VAR_OUTPUT
	stErr : ST_SiftError;
END_VAR

IF pJsonBuffer = 0 THEN
	stErr.bError := TRUE;
	stErr.nErrId := GVL_SIFT.NULL_JSON_POINTER;
	stErr.sReason := 'The JSON buffer is null';
	RETURN;
END_IF

fbJson.StartObject();

fbJson.AddKey('api_key');
fbJson.AddString(sApiKey);

fbJson.AddKey('grpc_uri');
fbJson.AddString(sGrpcUri);

fbJson.EndObject();

pJsonString := pJsonBuffer;
nBytes := fbJson.CopyDocument(pJsonString^, nLength);
IF nBytes = 0 THEN
	stErr.nErrId := GVL_SIFT.JSON_CAPACITY_REACHED;
	stErr.bError := TRUE;
	stErr.sReason := CONCAT(
		CONCAT('JSON msg too large: ', UDINT_TO_STRING(fbJson.GetDocumentLength())),
		' endpoint=authenticate',
	);
	RETURN;
END_IF

stErr := _F_CreateEndpointMessage(sEndpoint:='authenticate', 
								  pData:=pJsonString, 
								  nLength:=nBytes-1, 
                                  nBufferLength := nLength, 
                                  stMsg:=stMsg);

END_FUNCTION

// ---- POUs/Services/FB_PingService.TcPOU
FUNCTION_BLOCK FB_PingService
VAR_INPUT
	hSiftClient : T_SiftClient;
	bExecute : BOOL;
END_VAR

VAR_OUTPUT
	bBusy : BOOL;
	bError : BOOL;
	nErrId : UDINT;
	bSuccess : BOOL;
	stSiftError : ST_SiftError;
END_VAR

VAR
	eState : (IDLE, SEND_MESSAGE, WAIT_FOR_RESPONSE, SUCCESS, FAILURE) := IDLE;
	fbSendSiftMessage : _FB_SendSiftMessage;
	stPingReq : _ST_SiftMessage;
	fbJson : FB_JsonDomParser;
	sResponse : STRING(GVL_SIFT.MAX_JSON_RESPONSE_SIZE);
	jsonDoc : SJsonValue;
END_VAR

CASE eState OF
	IDLE:
		IF bExecute THEN
			eState := SEND_MESSAGE;
		END_IF
		
	SEND_MESSAGE:
		bBusy := TRUE;
		bError := FALSE;
		
		stSiftError := _F_CreatePingMessage(stMsg:=stPingReq);
		IF stSiftError.bError THEN
			nErrId := stSiftError.nErrId;
			eState := FAILURE;
		END_IF
		
		fbSendSiftMessage(hSiftClient:=hSiftClient, stMsg:=stPingReq, bExecute:=TRUE);
		eState := WAIT_FOR_RESPONSE;

	WAIT_FOR_RESPONSE:
		bBusy := TRUE;
		bError := FALSE;
		fbSendSiftMessage(bExecute:=FALSE);
		
		IF fbSendSiftMessage.bBusy THEN
			RETURN;
		ELSIF fbSendSiftMessage.bError THEN
			nErrId := GVL_SIFT.SIFT_PROXY_NO_RESPONSE;
			eState := FAILURE;
			RETURN;
		END_IF

		// Verify response.
		IF fbSendSiftMessage.stResponse.nLength > GVL_SIFT.MAX_JSON_RESPONSE_SIZE THEN
			nErrId := GVL_SIFT.JSON_CAPACITY_REACHED;
			eState := FAILURE;
			RETURN;	
		END_IF
		
		IF NOT SAFE_MEMCPY(ADR(sResponse), SIZEOF(sResponse), 
			               ADR(fbSendSiftMessage.stResponse.aData), fbSendSiftMessage.stResponse.nLength) THEN
			nErrId := GVL_SIFT.MEMCPY_ERROR;
			eState := FAILURE;
		END_IF
		
		jsonDoc := fbJson.ParseDocument(sResponse);
		
		IF _F_IsSuccessfulResponse(jsonDoc) THEN
			eState := SUCCESS;
		ELSE
			IF NOT _F_SetSiftError(jsonDoc, stSiftError) THEN
				nErrId := GVL_SIFT.SIFT_PROXY_INVALID_RESPONSE;
			END_IF
			nErrId := stSiftError.nErrId;
			eState := FAILURE;
		END_IF
		
	SUCCESS:
		bBusy := FALSE;
		bError := FALSE;
		bSuccess := TRUE;
		eState := IDLE;
		
	FAILURE:
		bBusy := FALSE;
		bError := TRUE;
		eState := IDLE;
END_CASE

END_FUNCTION_BLOCK

// ---- POUs/Services/FB_RunService.TcPOU
FUNCTION_BLOCK FB_RunService
VAR_INPUT
	hSiftClient : T_SiftClient;
	bExecute : BOOL;
	sName : STRING(255);
	sDescription : STRING(255);
	aTags : ARRAY[0..SiftClientParameters.MAX_NUM_TAGS - 1] OF STRING(255);
END_VAR

VAR_OUTPUT
	sId : STRING(255);
	bBusy : BOOL;
	bError : BOOL;
	nErrId : UDINT;
	stSiftError : ST_SiftError;
END_VAR

VAR
	eState : (IDLE, SEND_MESSAGE, WAIT_FOR_RESPONSE, SUCCESS, FAILURE) := IDLE;
	fbSendSiftMessage : _FB_SendSiftMessage;
	stRunReq : _ST_SiftMessage;
	fbJson : FB_JsonDomParser;
	sResponse : STRING(GVL_SIFT.MAX_JSON_RESPONSE_SIZE);
	jsonDoc : SJsonValue;	
END_VAR

CASE eState OF
	IDLE:
		IF bExecute THEN
			eState := SEND_MESSAGE;
		END_IF
		
	SEND_MESSAGE:
		bBusy := TRUE;
		bError := FALSE;
		
		stSiftError := _F_CreateRunMessage(stMsg:=stRunReq,
										   sName := sName,
										   sDescription := sDescription,
										   aTags := aTags,
										   pJsonBuffer := hSiftClient.pJsonBuffer,
										   nLength := hSiftClient.pJbLength);
		IF stSiftError.bError THEN
			nErrId := stSiftError.nErrId;
			eState := FAILURE;
		END_IF
		
		fbSendSiftMessage(hSiftClient:=hSiftClient, stMsg:=stRunReq, bExecute:=TRUE);
		eState := WAIT_FOR_RESPONSE;

	WAIT_FOR_RESPONSE:
		bBusy := TRUE;
		bError := FALSE;
		fbSendSiftMessage(bExecute := FALSE);
		
		IF fbSendSiftMessage.bBusy THEN
			RETURN;
		ELSIF fbSendSiftMessage.bError THEN
			nErrId := fbSendSiftMessage.nErrId;
			eState := FAILURE;
			RETURN;
		END_IF
		
		// Verify response.
		IF fbSendSiftMessage.stResponse.nLength > GVL_SIFT.MAX_JSON_RESPONSE_SIZE THEN
			nErrId := GVL_SIFT.JSON_CAPACITY_REACHED;
			eState := FAILURE;
			RETURN;	
		END_IF
		
		IF NOT SAFE_MEMCPY(ADR(sResponse), SIZEOF(sResponse), 
			               ADR(fbSendSiftMessage.stResponse.aData), fbSendSiftMessage.stResponse.nLength) THEN
			nErrId := GVL_SIFT.MEMCPY_ERROR;
			eState := FAILURE;
		END_IF
		
		jsonDoc := fbJson.ParseDocument(sResponse);
		IF jsonDoc = 0 THEN
			eState := FAILURE;
			nErrId := GVL_SIFT.UNABLE_TO_PARSE_JSON;
		END_IF
		
		IF _F_IsSuccessfulResponse(jsonDoc) THEN
			IF NOT fbJson.HasMember(jsonDoc, 'data') THEN
				nErrId := GVL_SIFT.SIFT_PROXY_INVALID_RESPONSE;
				eState := FAILURE;
				RETURN;
			END_IF
			jsonDoc := fbJson.FindMember(jsonDoc, 'data');
			
			IF NOT fbJson.HasMember(jsonDoc, 'run') THEN
				nErrId := GVL_SIFT.SIFT_PROXY_INVALID_RESPONSE;
				eState := FAILURE;
				RETURN;
			END_IF
			
			jsonDoc := fbJson.FindMember(jsonDoc, 'run');
			IF NOT fbJson.HasMember(jsonDoc, 'runId') THEN
				nErrId := GVL_SIFT.SIFT_PROXY_INVALID_RESPONSE;
				eState := FAILURE;
				RETURN;
			END_IF
			
			jsonDoc := fbJson.FindMember(jsonDoc, 'runId');
			sId := fbJson.GetString(jsonDoc);
			
			eState := SUCCESS;
		ELSE
			IF NOT _F_SetSiftError(jsonDoc, stSiftError) THEN
				nErrId := GVL_SIFT.SIFT_PROXY_INVALID_RESPONSE;
			END_IF
			nErrId := stSiftError.nErrId;
			eState := FAILURE;
		END_IF
		
	SUCCESS:
		bBusy := FALSE;
		bError := FALSE;
		eState := IDLE;
		
	FAILURE:
		bBusy := FALSE;
		bError := TRUE;
		eState := IDLE;
END_CASE

END_FUNCTION_BLOCK

// ---- POUs/Util/GetCurrentTime.TcPOU
// Returns a Sift compatible UTC timestamp. Should be used with FB_Ingest.WriteData().
FUNCTION GetCurrentTime : _ST_Timestamp
VAR_INPUT
END_VAR
VAR
	nUnixTimeNs : ULINT;
END_VAR

// Convert to UTC.
nUnixTimeNs := (F_GetSystemTime() - 116444736000000000) * 100;
GetCurrentTime.nSeconds := ULINT_TO_LINT(nUnixTimeNs/1_000_000_000);
GetCurrentTime.nNanoseconds := ULINT_TO_DINT(nUnixTimeNs MOD 1_000_000_000);

END_FUNCTION
